(* PLC project Unnamed, Unknown Unnamed 1 *)
(* stored: creationDateTime 2026-05-04T11:37:49, modificationDateTime 2026-05-04T11:37:49 *)

PROGRAM main
  VAR_INPUT
    Input1 : BOOL;
    Input2 : BOOL;
    Start : BOOL;
    Stop : BOOL;
  END_VAR
  VAR_OUTPUT
    Output1 : BOOL;
    Output2 : BOOL;
    Motor : BOOL;
  END_VAR

            Output1 := Input1 AND Input2;

(* This turns Output1 ON only when both Input1 AND Input2 are ON *)
(* Like a safety interlock - both doors must be closed before motor starts *)

(* OR Logic - Output2 turns ON when EITHER Input1 OR Input2 is ON *)
Output2 := Input1 OR Input2;

(* Latch circuit - START button turns motor on, STOP turns it off *)
(* Motor holds itself on even after START is released *)
IF Start AND NOT Stop THEN
    Motor := TRUE;
ELSIF Stop THEN
    Motor := FALSE;
END_IF;
          
END_PROGRAM

CONFIGURATION Config0
  RESOURCE Res0 ON PLC
    TASK task0(INTERVAL := T#20ms, PRIORITY := 1);
    PROGRAM instance0 WITH task0 : main;
  END_RESOURCE
END_CONFIGURATION
